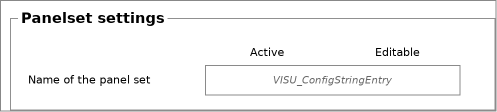
VISUALIZATION VISU_CoverConfig_PanelSet  // 497x112
VAR_IN_OUT
	activeConfig : CoverPanelSetConfig;
	editableConfig : CoverPanelSetConfig;
END_VAR
    GroupBox (10,10 485x100), "Panelset settings"
        Label (325,30 125x25), "Editable"
        Label (195,30 125x25), "Active"
        Frame (195,55 255x30)
            shows VISU_ConfigStringEntry(active := activeConfig.name, editable := editableConfig.name)
        Label (15,55 175x30), "Name of the panel set"
END_VISUALIZATION

(* stored: Version 1.1.0.1, ProductVersion 3.1.4019.2
   Visu VISU_CoverConfig_PanelSet: Id {73124879-1cb5-40fa-8831-61d4066865e3} *)
